// TIA Portal V21 export
VAR_GLOBAL   // PLC tag table "Cabinet_Config"
   M_Power_line_3_4_Available AT %M100.0 : Bool;
   M_Power_line_5_6_Available AT %M100.1 : Bool;
   M_Safety_zone_3_4_Available AT %M101.0 : Bool;
   M_Safety_zone_5_6_Available AT %M101.1 : Bool;
   M_Safety_zone_7_8_Available AT %M101.2 : Bool;
   M_Fast_doors_Enabled AT %M102.0 : Bool;
   M_Wrapping_machine_Enabled AT %M102.1 : Bool;
   M_CabinetNumberOutOfRange AT %M110.0 : Bool;
   M_HWCombiNumberOutOfRange AT %M110.1 : Bool;
END_VAR
VAR_GLOBAL CONSTANT   // user constants
   K_MaxCabinetNumber : UInt := 10;   // Max. number of C0 cabinets allowed
   K_MaxHWCombiNumber : UInt := 16;   // Max. number of defined PLC hardware combinations
END_VAR
